Fanuc KAREL source: kb00096.KL

-- PROVISIONAL review KL for V770-1; original PC SHA256 4cfbbc490d7be33add8792fbbb8bf9f297e9c105954974e86ad3e5f08f2a5c64
-- Incomplete behavior may be omitted. Consult companion uncertainty JSON. Do not deploy.
PROGRAM KB00096
%NOLOCKGROUP
BEGIN
  -- UNRESOLVED_PC offsets 5-12; opcodes 9D,23
  -- UNRESOLVED_PC offsets 17-24; opcodes 9D,23
  -- UNRESOLVED_PC offsets 29-36; opcodes 9D,23
  -- UNRESOLVED_PC offsets 41-52; opcodes 2E,23
  -- UNRESOLVED_PC offsets 57-66; opcodes 3F,75
  -- UNRESOLVED_PC offsets 71-78; opcodes 9D,23
  -- UNRESOLVED_PC offsets 83-125; opcodes 27,22,22,22,22,22,2A,22,31
  -- UNRESOLVED_PC offsets 130-134; opcodes 7F
END KB00096
